FUNCTION_BLOCK REAL2REAL
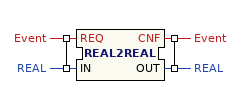
  EVENT_INPUT
    REQ WITH IN; (* Normal Execution Request *)
  END_EVENT
  EVENT_OUTPUT
    CNF WITH OUT; (* Execution Confirmation *)
  END_EVENT
  VAR_INPUT
    IN : REAL;
  END_VAR
  VAR_OUTPUT
    OUT : REAL;
  END_VAR
END_FUNCTION_BLOCK
